ABB RobotStudio station: ABB_Project_EGM_Stream_Control_Multiple.rspag

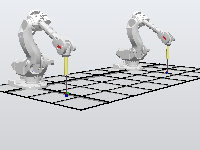
--- station ---
Station ABB_Project_EGM_Control_Type_2 (saved by RobotStudio 21.2.9526.0)
Controller Controller1
  mechanical unit ROB_1: IRB7600_325_310_Master, 6 joints, base frame (0, 0, 0) mm
  mechanical unit ROB_2: IRB7600_325_310_Slave, 6 joints, base frame (0, 5000, 0) mm
Layout (positions relative to the parent item):
  - IRB7600_325_310_Master [mechanism, from Robots\IRB7600_325_310_G_03.rslib] at (0, 0, 0) mm; joint values [-0.1606, -0.0866, 0.5233, 0, 1.1341, -0.1606] (rad or m)
  - IRB7600_325_310_Slave [mechanism, from Robots\IRB7600_325_310_G_03.rslib] at (0, 5000, 0) mm; joint values [-0.1606, -0.0866, 0.5233, 0, 1.1341, -0.1606] (rad or m)
  - ABB_GRIPPER_Master [mechanism, from Desktop\ABB_GRIPPER_Master.rslib] at (1773.65, -287.31, 1092.37) mm, rotated rx -180 ry 0 rz 180 deg
  - ABB_GRIPPER_Slave [mechanism] at (1773.65, 4712.69, 1092.37) mm, rotated rx -180 ry 0 rz 180 deg
      TCP ABB_GRIPPER at (0, 0, 1000) mm
      links: abb_gripper_2
Attachment: ABB_GRIPPER_Master is attached to IRB7600_325_310_Master / Link6
Attachment: ABB_GRIPPER_Slave is attached to IRB7600_325_310_Slave / Link6
Targets, tools, work objects and paths stored in the station and not in the controller backup, written as RAPID:
! task T_ROB1
MODULE Module1
  CONST robtarget Target_10:=[[1773.640630021,-268.046435456,592.370140835],[0.000008778,-0.000001192,-1,0.000000695],[-1,-1,-1,0],[9E+09,9E+09,9E+09,9E+09,9E+09,9E+09]];
  PROC Path_10()
    MoveL Target_10,v1000,z100,ABB_GRIPPER\WObj:=wobj0;
  ENDPROC
ENDMODULE

! task T_ROB2
MODULE Module1
  CONST robtarget Target_10:=[[1773.603022355,4713.049126298,577.782636007],[0.000003948,0.000001729,1,-0.000002752],[-1,-1,-1,0],[9E+09,9E+09,9E+09,9E+09,9E+09,9E+09]];
  LOCAL PERS wobjdata home_wobj:=[FALSE,TRUE,"",[[0,5000,0],[1,0,0,0]],[[0,0,0],[1,0,0,0]]];
  PROC Path_20()
    MoveL Target_10,v1000,z100,ABB_GRIPPER\WObj:=wobj0;
  ENDPROC
ENDMODULE


--- Backups/Controller1/RAPID/TASK1/PROGMOD/CalibData.mod ---
MODULE CalibData
    PERS tooldata ABB_GRIPPER:=[TRUE,[[0,0,1000],[1,0,0,0]],[10,[0,0.001,267.303],[1,0,0,0],0,0,0]];
ENDMODULE

--- Backups/Controller1/RAPID/TASK1/PROGMOD/Module1.mod ---
MODULE Module1
    ! Targets
    CONST robtarget P1 := [[1773.63,-287.31,92.37],[8.75873E-06,-1.19983E-06,-1,6.96016E-07],[-1,0,-1,0],[9E+09,9E+09,9E+09,9E+09,9E+09,9E+09]];
    CONST robtarget P2 := [[1380.38,1119.81,64.77],[2.64893E-05,0.0181086,-0.999836,1.00795E-05],[0,-1,0,0],[9E+09,9E+09,9E+09,9E+09,9E+09,9E+09]];
    CONST robtarget P3 := [[2043.85,1000.43,-65.59],[3.11237E-05,-2.11287E-06,-1,6.22279E-06],[0,-1,1,0],[9E+09,9E+09,9E+09,9E+09,9E+09,9E+09]];
    CONST robtarget P4 := [[1359.12,-183.33,35.71],[1.11593E-05,-4.04865E-06,-1,-3.67682E-06],[-1,0,-1,0],[9E+09,9E+09,9E+09,9E+09,9E+09,9E+09]];
    CONST robtarget P5 := [[1773.66,-287.32,35.72],[5.71756E-06,-4.42319E-06,-1,-3.51103E-07],[-1,0,-1,0],[9E+09,9E+09,9E+09,9E+09,9E+09,9E+09]];
    CONST robtarget P6 := [[2046.76,-166.95,92.34],[3.47833E-05,1.92386E-06,-1,-6.87548E-06],[-1,0,0,0],[9E+09,9E+09,9E+09,9E+09,9E+09,9E+09]];
    CONST robtarget P7 := [[2179.22,256.64,92.38],[1.67054E-05,3.20947E-05,-1,-5.605E-06],[0,-1,0,0],[9E+09,9E+09,9E+09,9E+09,9E+09,9E+09]];
    CONST robtarget P8 := [[1773.65,-287.31,92.39],[1.04985E-05,-1.1174E-06,-1,-1.91062E-07],[-1,0,-1,0],[9E+09,9E+09,9E+09,9E+09,9E+09,9E+09]];

    CONST robtarget P{8} := [P1, P2, P3, P4, P5, P6, P7, P8];

    ! Identifier for the EGM correction
    LOCAL VAR egmident egm_id;

    ! Actual State {Main State-Machine)
    VAR num actual_state := 0;
    ! Index of the Path
    VAR num p_index := 0;

    ! Initialization Parameters
    CONST num speed_tcp    := 50;
    CONST num speed_orient := 50;
    CONST speeddata speed_value := [speed_tcp,speed_orient,0,0];
    CONST zonedata zone_value := fine;

    ! Description:                                          !
    ! Simple movements with EGM Streaming Pos. - Main Cycle !
    PROC Main()
        TEST actual_state
            CASE 0:
                ! Register an EGM id
                EGMGetId egm_id;
                ! Setup the EGM communication
                EGMSetupUC ROB_1, egm_id, "default", "ROB_1";
                ! Start the EGM communication session
                EGMStreamStart egm_id \SampleRate:=4;

                ! Wait Time (2s)
                WaitTime 2;

                actual_state := 1;
            CASE 1:
                FOR i FROM 1 TO Dim(P, 1) DO
                    ! Move to the starting position for a point in index {n}
                    MoveJ P{i}, v200, fine, ABB_GRIPPER\WObj:=wobj0;

                    ! Wait Time (2s)
                    WaitTime 2;
                    ! Instructions for multiple movements for a point in index {n}
                    Path_Experiment_1 P{i}, speed_value, zone_value;
                    ! Wait Time (2s)
                    WaitTime 2;

                    ! Increase in value after a successfully executed path for a point in index {n}
                    p_index := p_index + 1;
                ENDFOR

                actual_state := 3;
            CASE 2:
                ! Instructions for multiple movements for a point in index {1}
                Path_Experiment_1 P{1}, speed_value, zone_value;
                ! Wait Time (2s)
                WaitTime 2;
                actual_state := 3;
            CASE 3:
                ! Move to the starting position
                MoveL P{1}, v200, fine, ABB_GRIPPER\WObj:=wobj0;

                actual_state := 4;
            CASE 4:
                ! Empty
        ENDTEST

        ! Stop and Release the EGM id
        !EGMStreamStop egm_id;
        !EGMReset egm_id;
    ENDPROC

    PROC Path_Experiment_1(robtarget rob_target, speeddata speed, zonedata zone)
        ! Block 1
        MoveL Offs (rob_target, 0, 300, 0), speed, zone, ABB_GRIPPER;
        MoveL rob_target, speed, zone, ABB_GRIPPER;
        MoveL Offs (rob_target, 0, 300, 0), v100, zone, ABB_GRIPPER;
        MoveL rob_target, v100, zone, ABB_GRIPPER;
        MoveL Offs (rob_target, 0, 300, 0), v500, zone, ABB_GRIPPER;
        MoveL rob_target, v500, zone, ABB_GRIPPER;
        ! Block 2
        MoveL Offs (rob_target, 300, 0, 0), speed, zone, ABB_GRIPPER;
        MoveL rob_target, speed, zone, ABB_GRIPPER;
        MoveL Offs (rob_target, 300, 0, 0), v100, zone, ABB_GRIPPER;
        MoveL rob_target, v100, zone, ABB_GRIPPER;
        MoveL Offs (rob_target, 300, 0, 0), v500, zone, ABB_GRIPPER;
        MoveL rob_target, v500, zone, ABB_GRIPPER;
        ! Block 3
        MoveL Offs (rob_target, 300, 300, 0), speed, zone, ABB_GRIPPER;
        MoveL rob_target, speed, zone, ABB_GRIPPER;
        MoveL Offs (rob_target, 300, 300, 0), v100, zone, ABB_GRIPPER;
        MoveL rob_target, v100, zone, ABB_GRIPPER;
        MoveL Offs (rob_target, 300, 300, 0), v500, zone, ABB_GRIPPER;
        MoveL rob_target, v500, zone, ABB_GRIPPER;
    ENDPROC
ENDMODULE

--- Backups/Controller1/RAPID/TASK2/PROGMOD/Module1.mod ---
MODULE Module1
    ! Identifier for the EGM correction
    LOCAL VAR egmident egm_id;
    ! EGM pose frames
    LOCAL CONST pose egm_correction_frame := [[0.0, 0.0, 0.0],[1.0, 0.0, 0.0, 0.0]];
    LOCAL CONST pose egm_sensor_frame     := [[0.0, 0.0, 0.0],[1.0, 0.0, 0.0, 0.0]];
    ! The work object. Base Frame
    LOCAL PERS wobjdata egm_wobj   := [FALSE,TRUE,"",[[0,5000,0],[1,0,0,0]],[[0,0,0],[1,0,0,0]]];
    ! Limits for convergence
    ! Cartesian: +- 0.1 mm
    LOCAL CONST egm_minmax egm_condition_cartesian := [-0.1, 0.1];
    ! Orientation: +- 0.1 degrees
    LOCAL CONST egm_minmax egm_condition_orient := [-0.1, 0.1];

    ! Initial targets of the Robot {Master}
    CONST robtarget P1 := [[1773.63,-287.31,92.37],[8.75873E-06,-1.19983E-06,-1,6.96016E-07],[-1,0,-1,0],[9E+09,9E+09,9E+09,9E+09,9E+09,9E+09]];
    CONST robtarget P2 := [[1380.38,1119.81,64.77],[2.64893E-05,0.0181086,-0.999836,1.00795E-05],[0,-1,0,0],[9E+09,9E+09,9E+09,9E+09,9E+09,9E+09]];
    CONST robtarget P3 := [[2043.85,1000.43,-65.59],[3.11237E-05,-2.11287E-06,-1,6.22279E-06],[0,-1,1,0],[9E+09,9E+09,9E+09,9E+09,9E+09,9E+09]];
    CONST robtarget P4 := [[1359.12,-183.33,35.71],[1.11593E-05,-4.04865E-06,-1,-3.67682E-06],[-1,0,-1,0],[9E+09,9E+09,9E+09,9E+09,9E+09,9E+09]];
    CONST robtarget P5 := [[1773.66,-287.32,35.72],[5.71756E-06,-4.42319E-06,-1,-3.51103E-07],[-1,0,-1,0],[9E+09,9E+09,9E+09,9E+09,9E+09,9E+09]];
    CONST robtarget P6 := [[2046.76,-166.95,92.34],[3.47833E-05,1.92386E-06,-1,-6.87548E-06],[-1,0,0,0],[9E+09,9E+09,9E+09,9E+09,9E+09,9E+09]];
    CONST robtarget P7 := [[2179.22,256.64,92.38],[1.67054E-05,3.20947E-05,-1,-5.605E-06],[0,-1,0,0],[9E+09,9E+09,9E+09,9E+09,9E+09,9E+09]];
    CONST robtarget P8 := [[1773.65,-287.31,92.39],[1.04985E-05,-1.1174E-06,-1,-1.91062E-07],[-1,0,-1,0],[9E+09,9E+09,9E+09,9E+09,9E+09,9E+09]];

    ! Description:                                !
    ! Externally Guided motion (EGM) - Main Cycle !
    PROC main()
        ! Move to the starting position
        !MoveL P1,v500,fine,ABB_GRIPPER\WObj:=egm_wobj;

        ! Call -> Cartesian Move Procedure (EGM)
        EGM_CARTESIAN_MOVE;
    ENDPROC

    PROC EGM_CARTESIAN_MOVE()
        ! Description:                                       !
        ! Externally Guided motion (EGM) - Cartesian Control !

        ! Register an EGM id
        EGMGetId egm_id;

        ! Setup the EGM communication
        EGMSetupUC ROB_2, egm_id, "default", "ROB_2", \Pose;

        ! EGM While {Cartesian}
        WHILE TRUE DO
            ! Prepare for an EGM communication session
            EGMActPose egm_id,
                       \Tool:=ABB_GRIPPER,
                       \WObj:=egm_wobj,
                       egm_correction_frame,
                       EGM_FRAME_BASE,
                       egm_sensor_frame,
                       EGM_FRAME_BASE
                       \X:=egm_condition_cartesian
                       \Y:=egm_condition_cartesian
                       \Z:=egm_condition_cartesian
                       \Rx:=egm_condition_orient
                       \Ry:=egm_condition_orient
                       \Rz:=egm_condition_orient
                       \LpFilter:=100
                       \SampleRate:=4
                       \MaxPosDeviation:=1000
                       \MaxSpeedDeviation:=100;

            ! Start the EGM communication session
            EGMRunPose egm_id, EGM_STOP_RAMP_DOWN, \X \Y \Z \Rx \Ry \Rz \CondTime:=2000 \RampInTime:=0.1 \RampOutTime:=0.1 \PosCorrGain:=1.0;
            ! Release the EGM id
            !EGMReset egm_id;
            ! Wait 2 seconds {No data from EGM sensor}
            !WaitTime 2;
        ENDWHILE

        ERROR
        IF ERRNO = ERR_UDPUC_COMM THEN
            TPWrite "Communication timedout";
            TRYNEXT;
        ENDIF
    ENDPROC
ENDMODULE
